//{attribute 'qualified_only'}
//{attribute 'strict'}
{attribute 'to_string'}
{attribute 'to_wstring'}
TYPE E_St040_Settings :
(
	//eSt040_Settings_none := 0,
	
	eSt040_Settings_Station_Deaktiv,	// Station deaktivieren
	eSt040_Settings_Autohome,			// automatic home with start button
	
	eSt040_Settings_JogSpeed,			// Tippgeschwindigkeit [mm/s]
	eSt040_Settings_WorkSpeed,			// Automatik-Geschwindigkeit  [mm/s]
	
	eSt040_Settings_PosHome,			// Homeposition [mm]
	eSt040_Settings_PosWork,			// Arbeitsposition [mm]
	
	eSt040_Settings_XPosStor1,			// Teach-Position, Storage 1 X [mm]
	eSt040_Settings_YPosStor1,			// Teach-Position, Storage 1 Y [mm]
	eSt040_Settings_ZPosStor1,			// Teach-Position, Storage 1 Z [mm]
	    
	eSt040_Settings_XPosStor2,			// Teach-Position, Storage 2 X [mm]
	eSt040_Settings_YPosStor2,			// Teach-Position, Storage 2 Y [mm]
	eSt040_Settings_ZPosStor2,			// Teach-Position, Storage 2 Z [mm]
	
	
	/// has to be set to last index for array bounds!
	eSt040_Settings_nMaxIdx	
);
END_TYPE

(* stored: Version 1.1.0.1
   DUT E_St040_Settings: Id {7188bc62-3d80-4e24-9ea3-015c3e25b39e} *)
